RoboDK station: movimiento_mocap14dic.rdk

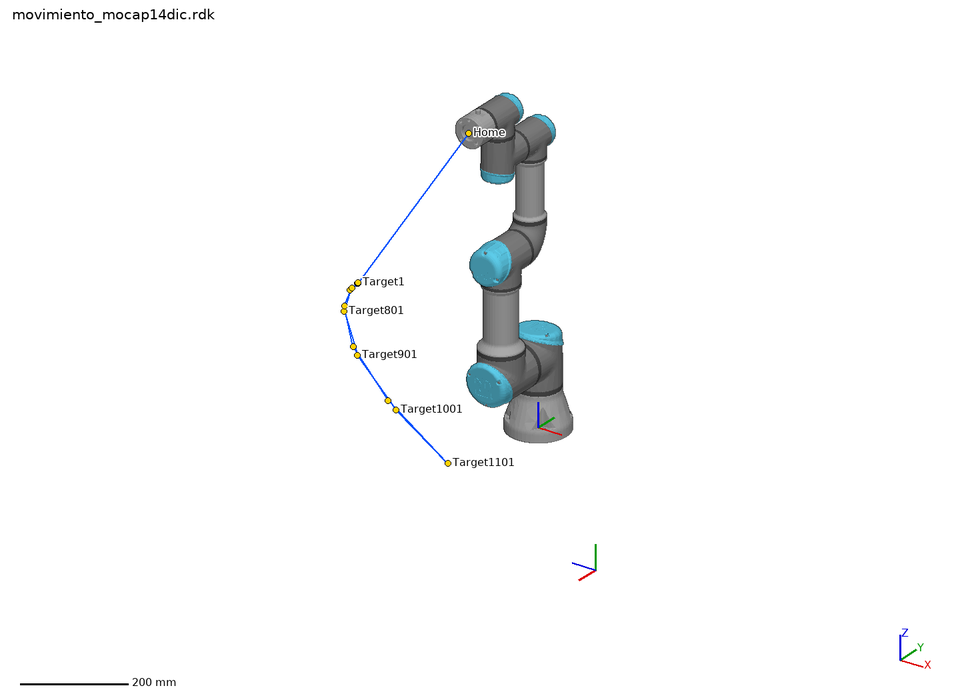
[picture v0: the station drawn from its stored meshes, robots at their saved joint values, targets as dots, program paths as lines]
Station movimiento_mocap (saved by RoboDK 5.5.2). Poses are relative to the parent item; angles as X-Y-Z fixed-axis rotations.
  - frame UR3e Base at (0, 0, 0) mm
    - robot UR3e: 6 axes, payload 3 kg, reach 500 mm, repeatability 0.03 mm, weight 11 kg
        modified DH rows (alpha deg, a mm, theta deg, d mm): 0, 0, 0, 151.9; 90, 0, 180, 0; 0, 243.55, 0, 0; 0, 213.2, 0, 131.05; -90, 0, 0, 85.35; 90, 0, 180, 92.1
        joint limits [-360, -360, -360, -360, -360, -360] to [360, 360, 360, 360, 360, 360]; home [0, -90, -90, 0, 90, 0]; saved at [0, -90, 0, -90, 0, 0]
    - frame B0 frame at (430, -430, 0) mm, rotated rx 90 ry 0 rz -90 deg
      - target Home (joint target) at (-206.85, 694, 430) mm, rotated rx 0 ry -90 rz -180 deg; joints [0, -90, 0, -90, 0, 0] of UR3e
      - target Target1 (Cartesian target) at (413.82, 686.35, 244.18) mm, rotated rx -178.32 ry -4.28 rz -12.94 deg; joints [0, -90, 0, -90, 0, 0] of UR3e
      - target Target101 (Cartesian target) at (413.88, 686.39, 244.05) mm, rotated rx -178.38 ry -3.98 rz -12.88 deg; joints [0, -90, 0, -90, 0, 0] of UR3e
      - target Target201 (Cartesian target) at (413.8, 686.33, 244.19) mm, rotated rx -178.32 ry -4.3 rz -12.96 deg; joints [0, -90, 0, -90, 0, 0] of UR3e
      - target Target301 (Cartesian target) at (413.88, 686.38, 244.04) mm, rotated rx -178.36 ry -4 rz -12.89 deg; joints [0, -90, 0, -90, 0, 0] of UR3e
      - target Target401 (Cartesian target) at (413.8, 686.35, 244.19) mm, rotated rx -178.34 ry -4.3 rz -12.99 deg; joints [0, -90, 0, -90, 0, 0] of UR3e
      - target Target501 (Cartesian target) at (413.79, 686.35, 244.19) mm, rotated rx -178.34 ry -4.32 rz -12.98 deg; joints [0, -90, 0, -90, 0, 0] of UR3e
      - target Target601 (Cartesian target) at (416.31, 686.44, 244.15) mm, rotated rx -178.31 ry -4.31 rz -13.65 deg; joints [0, -90, 0, -90, 0, 0] of UR3e
      - target Target701 (Cartesian target) at (443.63, 684.39, 241.2) mm, rotated rx -178.61 ry -4.53 rz -18.67 deg; joints [0, -90, 0, -90, 0, 0] of UR3e
      - target Target801 (Cartesian target) at (495.71, 668.07, 218.57) mm, rotated rx -2.72 ry -1.11 rz -15.08 deg; joints [0, -90, 0, -90, 0, 0] of UR3e
      - target Target901 (Cartesian target) at (546.59, 615.77, 152.81) mm, rotated rx -12.96 ry -4.21 rz -26.44 deg; joints [0, -90, 0, -90, 0, 0] of UR3e
      - target Target1001 (Cartesian target) at (549.78, 530.02, 63.34) mm, rotated rx -29.12 ry -9.56 rz -32.07 deg; joints [0, -90, 0, -90, 0, 0] of UR3e
      - target Target1101 (Cartesian target) at (496.45, 421.8, -15.74) mm, rotated rx 131.92 ry -26.26 rz -33.84 deg; joints [0, -90, 0, -90, 0, 0] of UR3e
      - target Target1201 (Cartesian target) at (553.05, 546.88, 79.21) mm, rotated rx -26.07 ry -8.34 rz -31.75 deg; joints [0, -90, 0, -90, 0, 0] of UR3e
      - target Target1301 (Cartesian target) at (540.12, 627.93, 166.97) mm, rotated rx 170.52 ry -9.23 rz -36.97 deg; joints [0, -90, 0, -90, 0, 0] of UR3e
      - target Target1401 (Cartesian target) at (485.41, 672.98, 225.11) mm, rotated rx 178.99 ry -5.23 rz -26.22 deg; joints [0, -90, 0, -90, 0, 0] of UR3e
      - target Target1501 (Cartesian target) at (436.94, 685.26, 242.46) mm, rotated rx -178.47 ry -4.35 rz -17.38 deg; joints [0, -90, 0, -90, 0, 0] of UR3e
      - target Target1601 (Cartesian target) at (414.5, 686.4, 244.18) mm, rotated rx -178.3 ry -4.29 rz -13.28 deg; joints [0, -90, 0, -90, 0, 0] of UR3e
      - target Target1701 (Cartesian target) at (413.79, 686.37, 244.17) mm, rotated rx -178.35 ry -4.3 rz -12.99 deg; joints [0, -90, 0, -90, 0, 0] of UR3e
      - target Target1801 (Cartesian target) at (413.8, 686.36, 244.18) mm, rotated rx -178.33 ry -4.3 rz -12.97 deg; joints [0, -90, 0, -90, 0, 0] of UR3e
  - program My Prog (20 instructions, listed below)
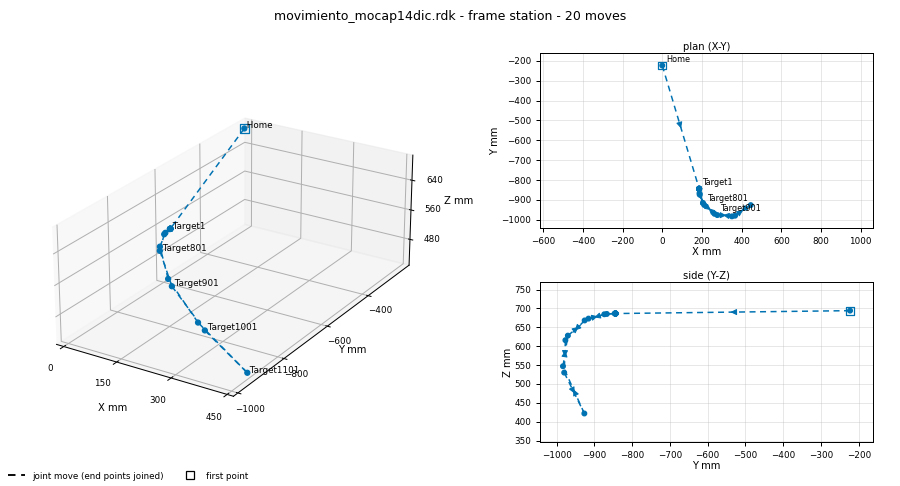
[picture p0: tool path of movimiento_mocap14dic.rdk in frame station, 20 of 20 moves have a stored position in this frame; points joined in program order, loops and branches not executed]

--- program My Prog (robot UR3e) ---
  MoveJ (Home)
  MoveJ (Target1)
  MoveJ (Target101)
  MoveJ (Target201)
  MoveJ (Target301)
  MoveJ (Target401)
  MoveJ (Target501)
  MoveJ (Target601)
  MoveJ (Target701)
  MoveJ (Target801)
  MoveJ (Target901)
  MoveJ (Target1001)
  MoveJ (Target1101)
  MoveJ (Target1201)
  MoveJ (Target1301)
  MoveJ (Target1401)
  MoveJ (Target1501)
  MoveJ (Target1601)
  MoveJ (Target1701)
  MoveJ (Target1801)
